TYPE T_AnyBit : __SYSTEM.AnyType; END_TYPE

(* stored: Version 1.1.0.1
   DUT T_AnyBit: Id {e1b57a9e-bd4c-493b-a67e-61064484fedf} *)
